FUNCTION_BLOCK Controller (* Basic Function Block Type *)
  (* Standard: 61499-2 *)
  (* Version 0.3, 2009-09-15, JHC, Holobloc Inc, Changed transition priorities. *)
  (* Version 0.2, 2003-12-04, JHC, Rockwell Automation, Renamed for better indexing. *)
  (* Version 0.1, 2002-11-05, JHC, Rockwell Automation, Corrected missing ST element in Algorithm REQ. *)
  (* Version 0.0, 2000-05-30, JHC, Rockwell Automation *)
  (* Compiler header: package fb.rt.template; *)
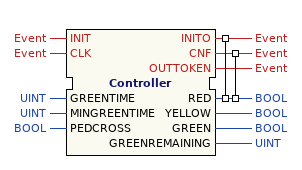
  EVENT_INPUT
    INIT; (* Initialization Request *)
    CLK; (* Normal Execution Request *)
  END_EVENT
  EVENT_OUTPUT
    INITO WITH RED; (* Initialization Confirm *)
    CNF WITH RED; (* Execution Confirmation *)
    OUTTOKEN;
  END_EVENT
  VAR_INPUT
    GREENTIME : UINT;
    MINGREENTIME : UINT;
    PEDCROSS : BOOL;
  END_VAR
  VAR_OUTPUT
    RED : BOOL; (* Output event qualifier *)
    YELLOW : BOOL;
    GREEN : BOOL;
    GREENREMAINING : UINT;
  END_VAR
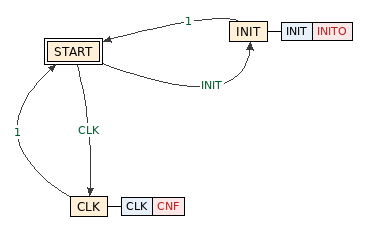
  EC_STATES
    START; (* Initial State *)
    INIT : INIT -> INITO; (* Initialization *)
    CLK : CLK -> CNF; (* Normal execution *)
  END_STATES
  EC_TRANSITIONS
    INIT TO START := 1;
    START TO CLK := CLK;
    START TO INIT := INIT;
    CLK TO START := 1;
  END_TRANSITIONS
  ALGORITHM INIT IN ST: (* Initialization algorithm *)
RED:=FALSE;
YELLOW:=FALSE;
GREEN:=FALSE;
GREENTIME:=0;
MINGREENTIME:=0;
PEDCROSS:=FALSE;
  END_ALGORITHM
  ALGORITHM CLK IN ST: (* Normally executed algorithm *)
GREENTIME:= GREENTIME - 1
  END_ALGORITHM
END_FUNCTION_BLOCK
